PROGRAM P_Demo_FB_JsonDomParser_GetHexBinary
VAR
    fbParser : FB_JsonDomParser; // 父 FB 实例
    v : SJsonValue;
    p : PVOID;
    n : DINT;
    vRet : DINT; // 返回值监视
    bTrigger : BOOL := FALSE; // 在线置 TRUE 触发一次调用
    bTriggerPrev : BOOL;
END_VAR

// =============================================================================
// 场景：从已解析的 JSON DOM 中读取某字段的 HexBinary 类型值（如解析云端下发指令里的目标速度、批次号、状态码）。
// 价值：按节点直接取值，比反复扫字符串快。
// 验证：登录 PLC 在线写 bTrigger := TRUE 触发，monitor 返回值/输出参数。具体步骤见下方注释。
// 验证步骤：
//   1. 右键 PLC 项目下 POUs 文件夹 → Add → Existing Item → 选本 .TcPOU 文件
//   2. 引用 Tc3_JsonXml（References → Add library）
//   3. 编译 → 登录 → 运行；按 verify 注释里给出的在线写值操作
// =============================================================================

// 上升沿触发一次方法调用并观察输出。
IF bTrigger AND NOT bTriggerPrev THEN
    vRet := fbParser.GetHexBinary(
        v := v,
        p := p,
        n := n
    );
END_IF;
bTriggerPrev := bTrigger;

END_PROGRAM

(* stored: Version 1.1.0.1, ProductVersion 3.1.4024.5
   POU P_Demo_FB_JsonDomParser_GetHexBinary: Id {a60a280f-bce0-5848-b30b-cda38856e82c}, SpecialFunc None *)
